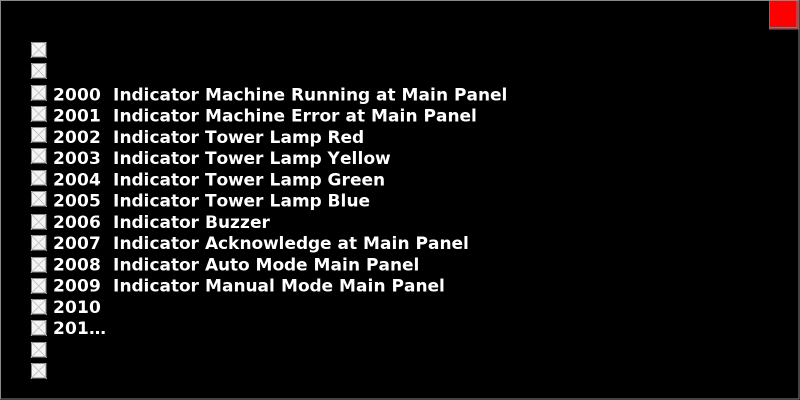
VISUALIZATION P1_DO1  // 800x400, background image 
    ImageSwitcher (31,42 15x15), variable: InputOutput_GVL.xIn1000, behaviour: TOGGLE
    Label (50,16 625x391), "2000 Indicator Machine Running at Main Panel 2001 Indicator Machine Error at Main Panel 2002 Indicator Tower Lamp Red 2003 Indicator Tower Lamp Yellow 2004 Indicator Tower Lamp Green 2005 Indicator Tower Lamp Blue 2006 Indicator Buzzer 2007 Indicator Acknowledge at Main Panel 2008 Indicator Auto Mode Main Panel 2009 Indicator Manual Mode Main Panel 2010 2011 2012 2013 2014 2015"
    ImageSwitcher (31,63 15x15), variable: InputOutput_GVL.xIn1001, behaviour: TOGGLE
    ImageSwitcher (31,85 15x15), variable: InputOutput_GVL.xIn1002, behaviour: TOGGLE
    ImageSwitcher (31,106 15x15), variable: InputOutput_GVL.xIn1003, behaviour: TOGGLE
    ImageSwitcher (31,127 15x15), variable: InputOutput_GVL.xIn1004, behaviour: TOGGLE
    ImageSwitcher (31,148 15x15), variable: InputOutput_GVL.xIn1005, behaviour: TOGGLE
    ImageSwitcher (31,170 15x15), variable: InputOutput_GVL.xIn1006, behaviour: TOGGLE
    ImageSwitcher (31,191 15x15), variable: InputOutput_GVL.xIn1007, behaviour: TOGGLE
    ImageSwitcher (31,214 15x15), variable: InputOutput_GVL.xIn1008, behaviour: TOGGLE
    ImageSwitcher (31,235 15x15), variable: InputOutput_GVL.xIn1009, behaviour: TOGGLE
    ImageSwitcher (31,257 15x15), variable: InputOutput_GVL.xIn1010, behaviour: TOGGLE
    ImageSwitcher (31,278 15x15), variable: InputOutput_GVL.xIn1011, behaviour: TOGGLE
    ImageSwitcher (31,299 15x15), variable: InputOutput_GVL.xIn1012, behaviour: TOGGLE
    ImageSwitcher (31,320 15x15), variable: InputOutput_GVL.xIn1013, behaviour: TOGGLE
    ImageSwitcher (31,342 15x15), variable: InputOutput_GVL.xIn1014, behaviour: TOGGLE
    ImageSwitcher (31,363 15x15), variable: InputOutput_GVL.xIn1015, behaviour: TOGGLE
    Button (769,-1 30x30), image: VisuSymbols.Symbols.Wrong
        OnMouseClick: CloseDialog Dialog=P1_DO1, Result=OK, NumpadKeypadSet=True
END_VISUALIZATION

(* stored: Version 1.1.0.1, ProductVersion 3.1.4024.12
   Visu P1_DO1: Id {2587e045-13f2-4a1d-9465-d812995e4207} *)
